// TIA Portal V20 export
ORGANIZATION_BLOCK "Main"   // OB1, LAD, ProgramCycle
TITLE = "Main Program Sweep (Cycle)"
// stored: AutoNumber false, IsIECCheckEnabled true, SetENOAutomatically true
   VAR_INPUT
      Initial_Call : Bool;   // Initial call of this OB
      Remanence : Bool;   // =True, if remanent data are available
   END_VAR
BEGIN

REGION Network 1: First Cycle
   // Set bit to true in first cycle, and false in all other cycles
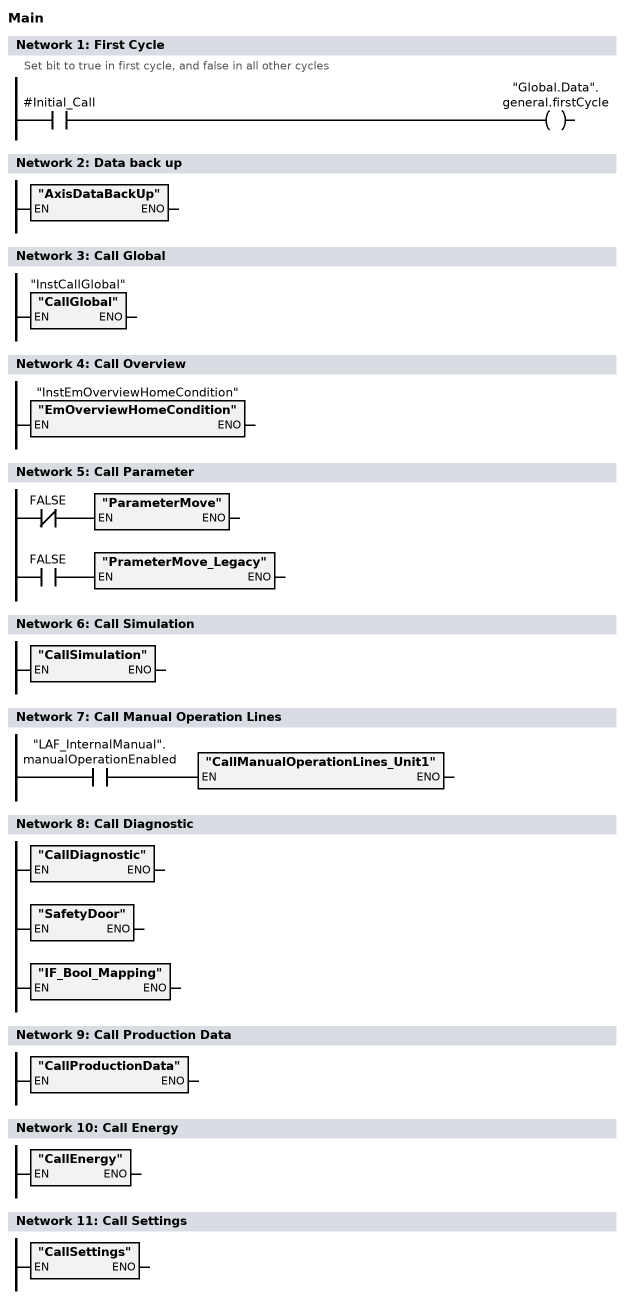
   RUNG wire#powerrail
      Contact( #Initial_Call )
      Coil( "Global.Data".general.firstCycle )
   END_RUNG
   // the same network as SCL:
   "Global.Data".general.firstCycle := #Initial_Call;
END_REGION

REGION Network 2: Data back up
   RUNG wire#powerrail
      "AxisDataBackUp"()
   END_RUNG
   // the same network as SCL:
   "AxisDataBackUp"();
END_REGION

REGION Network 3: Call Global
   RUNG wire#powerrail
      "InstCallGlobal"()
   END_RUNG
   // the same network as SCL:
   "InstCallGlobal"();   // "CallGlobal"
END_REGION

REGION Network 4: Call Overview
   RUNG wire#powerrail
      "InstEmOverviewHomeCondition"()
   END_RUNG
   // the same network as SCL:
   "InstEmOverviewHomeCondition"();   // "EmOverviewHomeCondition"
END_REGION

REGION Network 5: Call Parameter
   RUNG wire#powerrail
      I_Contact( FALSE )
      "ParameterMove"()
   END_RUNG
   RUNG wire#powerrail
      Contact( FALSE )
      "PrameterMove_Legacy"()
   END_RUNG
   // the same network as SCL:
   IF NOT FALSE THEN "ParameterMove"(); END_IF;
   IF FALSE THEN "PrameterMove_Legacy"(); END_IF;
END_REGION

REGION Network 6: Call Simulation
   RUNG wire#powerrail
      "CallSimulation"()
   END_RUNG
   // the same network as SCL:
   "CallSimulation"();
END_REGION

REGION Network 7: Call Manual Operation Lines
   RUNG wire#powerrail
      Contact( "LAF_InternalManual".manualOperationEnabled )
      "CallManualOperationLines_Unit1"()
   END_RUNG
   // the same network as SCL:
   IF "LAF_InternalManual".manualOperationEnabled THEN "CallManualOperationLines_Unit1"(); END_IF;
END_REGION

REGION Network 8: Call Diagnostic
   RUNG wire#powerrail
      "CallDiagnostic"()
   END_RUNG
   RUNG wire#powerrail
      "SafetyDoor"()
   END_RUNG
   RUNG wire#powerrail
      "IF_Bool_Mapping"()
   END_RUNG
   // the same network as SCL:
   "CallDiagnostic"();
   "SafetyDoor"();
   "IF_Bool_Mapping"();
END_REGION

REGION Network 9: Call Production Data
   RUNG wire#powerrail
      "CallProductionData"()
   END_RUNG
   // the same network as SCL:
   "CallProductionData"();
END_REGION

REGION Network 10: Call Energy
   RUNG wire#powerrail
      "CallEnergy"()
   END_RUNG
   // the same network as SCL:
   "CallEnergy"();
END_REGION

REGION Network 11: Call Settings
   RUNG wire#powerrail
      "CallSettings"()
   END_RUNG
   // the same network as SCL:
   "CallSettings"();
END_REGION
END_ORGANIZATION_BLOCK
